FUNCTION_BLOCK EQUIP_VisionSensor (* Composite Function Block Type *)
  (* Standard: 61499-2 *)
  (* Version 0.0, 08/01/2026, Schneider Electric, template *)
  PACKAGE Main;
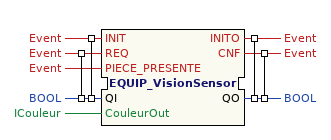
  EVENT_INPUT
    INIT WITH QI; (* Initialization Request *)
    REQ WITH QI; (* Normal Execution Request *)
    PIECE_PRESENTE;
  END_EVENT
  EVENT_OUTPUT
    INITO WITH QO; (* Initialization Confirm *)
    CNF WITH QO; (* Execution Confirmation *)
  END_EVENT
  VAR_INPUT
    QI : BOOL; (* Input event qualifier *)
  END_VAR
  VAR_OUTPUT
    QO : BOOL; (* Output event qualifier *)
  END_VAR
  SOCKETS
    CouleurOut : ICouleur; (* Sortie couleur *)
  END_SOCKETS
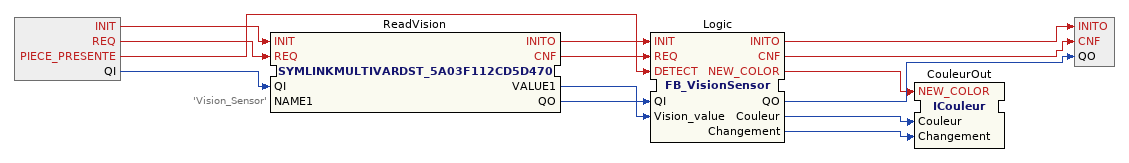
  FBS
    ReadVision : SYMLINKMULTIVARDST_5A03F112CD5D470(NAME1 := 'Vision_Sensor'); {SET_ATTRIBUTE(Configuration.GenericFBType.InterfaceParams, Runtime.System#I:=1;VALUE${I$}:INT)}
    Logic : FB_VisionSensor;
  END_FBS
  EVENT_CONNECTIONS
    Logic.INITO TO INITO;
    Logic.CNF TO CNF;
    PIECE_PRESENTE TO Logic.DETECT;
    Logic.NEW_COLOR TO CouleurOut.NEW_COLOR;
    INIT TO ReadVision.INIT;
    REQ TO ReadVision.REQ;
    ReadVision.INITO TO Logic.INIT;
    ReadVision.CNF TO Logic.REQ;
  END_CONNECTIONS
  DATA_CONNECTIONS
    Logic.Couleur TO CouleurOut.Couleur;
    Logic.Changement TO CouleurOut.Changement;
    QI TO ReadVision.QI;
    ReadVision.VALUE1 TO Logic.Vision_value;
    Logic.QO TO QO;
    ReadVision.QO TO Logic.QI;
  END_CONNECTIONS
END_FUNCTION_BLOCK
